(* CODESYS project Ladder1.project

Project tree, tasks and I/O mapping:
  Device : CODESYS Control Win V3, 3S - Smart Software Solutions GmbH, order no. 305021, version 3.5.10.30
    application Application
      libraries: Standard, * (System)
      task MainTask (cyclic, interval t#20ms, priority 1) calls PLC_PRG
      task VISU_TASK (cyclic, interval 100 ms, priority 31) calls VisuElems.Visu_Prg
      program PLC_PRG [LD]
      visualisation Visualization1
  libraries: VisuSymbols, 3.5.10.0 (System)
  text list GlobalTextList
*)

// Device/Application/PLC_PRG
PROGRAM PLC_PRG
VAR
	Contact1: BOOL := FALSE;
	Coil1: BOOL;
	Contact2: BOOL := FALSE;
	Contact3: BOOL := TRUE;
END_VAR

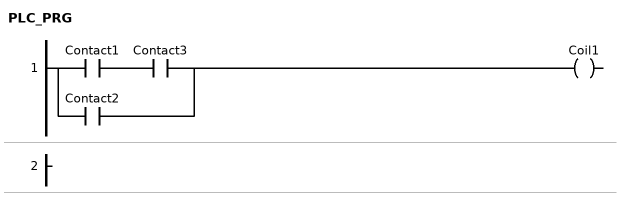
// NETWORK 1
Coil1 := Contact1 AND Contact3 OR Contact2;

// NETWORK 2

END_PROGRAM

// Device/Application/Visualization1
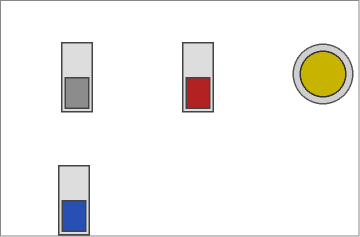
VISUALIZATION Visualization1  // 360x237
    DipSwitch (42,42 70x70), variable: PLC_PRG.Contact1, behaviour: TOGGLE, style: Switch-DipSwitch-Gray
    Lamp1 (288,39 70x70), variable: PLC_PRG.Coil1, style: Lamp-Lamp1-Yellow
    DipSwitch (39,165 70x70), variable: PLC_PRG.Contact2, behaviour: TOGGLE, style: Switch-DipSwitch-Blue
    DipSwitch (163,42 70x70), variable: PLC_PRG.Contact3, behaviour: TOGGLE, style: Switch-DipSwitch-Red
END_VISUALIZATION
